PROGRAM MAIN
VAR
END_VAR

POU_COMM();
POU_IN();
POU_CNTRL_M1_AUX();
POU_CNTRL_M1();
POU_OUT();

END_PROGRAM

(* stored: Version 1.1.0.1
   POU MAIN: Id {09203c6b-b88c-470c-8b16-8e729a6797e5}, SpecialFunc None *)
